// Device/Application/F020_HMI_Pages/F020_PartX_Screen
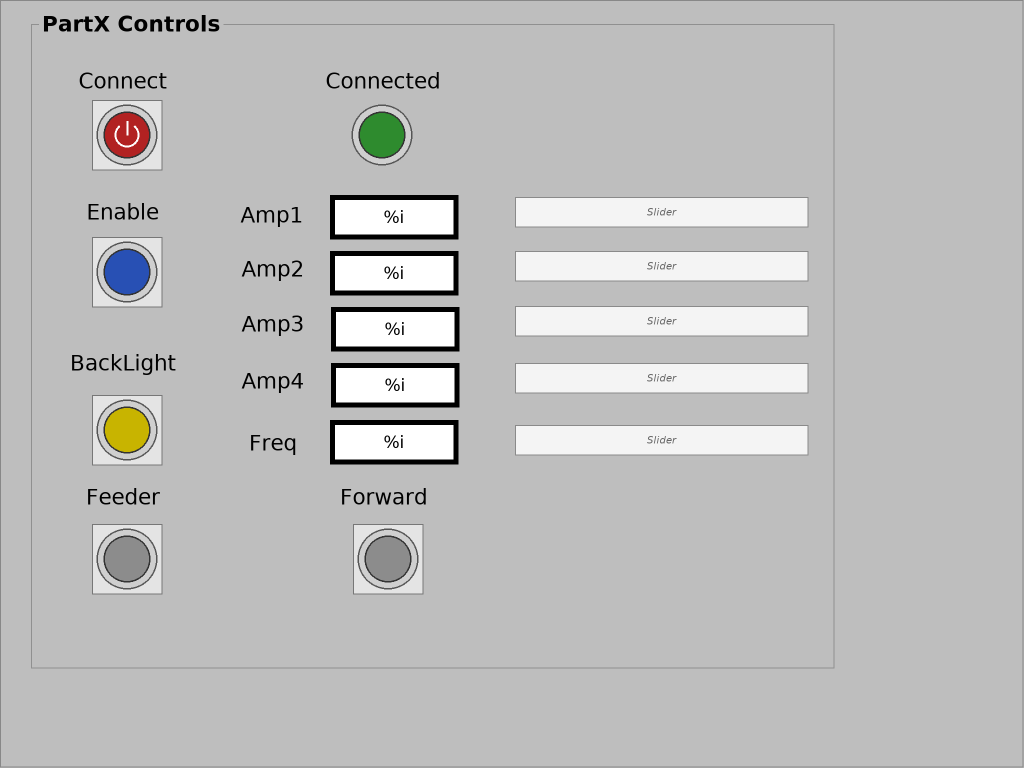
VISUALIZATION F020_PartX_Screen  // 1024x768
    GroupBox (31,16 803x652), "PartX Controls"
        Label (17,50 150x30), "Connect"
        PushSwitch (61,221 70x70), variable: GVL.PARTX.MAN, behaviour: TOGGLE, style: Switch-PushSwitch-Blue
        PowerSwitch (61,84 70x70), variable: GVL.PARTX.ENABLE_TCP, behaviour: TOGGLE, style: Switch-PowerSwitch-Red
        Label (17,181 150x30), "Enable"
        Textfield (299,179 128x44), "%i", text variable: GVL.PARTX.Amp1
            OnMouseClick: write the text variable via VisuDialogs.Numpad
        Label (277,50 150x30), "Connected"
        Label (166,184 150x30), "Amp1"
        Lamp1 (316,84 70x70), variable: F002_SR02_SOCKET_CLIENT.Client.xActive, style: Lamp-Lamp1-Green
        Textfield (299,235 128x44), "%i", text variable: GVL.PARTX.Amp2
            OnMouseClick: write the text variable via VisuDialogs.Numpad
        PushSwitch (61,379 70x70), variable: GVL.PARTX.BackLight, behaviour: TOGGLE, style: Switch-PushSwitch-Yellow
        Label (17,332 150x30), "BackLight"
        Label (167,238 150x30), "Amp2"
        Textfield (300,291 128x44), "%i", text variable: GVL.PARTX.Amp3
            OnMouseClick: write the text variable via VisuDialogs.Numpad
        Label (167,293 150x30), "Amp3"
        Textfield (300,347 128x44), "%i", text variable: GVL.PARTX.Amp4
            OnMouseClick: write the text variable via VisuDialogs.Numpad
        Label (167,350 150x30), "Amp4"
        Textfield (299,404 128x44), "%i", text variable: GVL.PARTX.Freq
            OnMouseClick: write the text variable via VisuDialogs.Numpad
        Label (167,412 150x30), "Freq"
        PushSwitch (61,508 70x70), variable: GVL.PARTX.Feeder_Enable, behaviour: TOGGLE, style: Switch-PushSwitch-Gray
        Label (17,466 150x30), "Feeder"
        Slider (484,181 293x30), variable: GVL.PARTX.Amp1, scale 0..100
        Slider (484,235 293x30), variable: GVL.PARTX.Amp2, scale 0..100
        Slider (484,290 293x30), variable: GVL.PARTX.Amp3, scale 0..100
        Label (278,466 150x30), "Forward"
        Label (472,466 150x30)
    Slider (515,363 293x30), variable: GVL.PARTX.Amp4, scale 0..100
    Slider (515,425 293x30), variable: GVL.PARTX.Freq, scale 0..100
    PushSwitch (353,524 70x70), variable: GVL.PARTX.FWD, behaviour: TOGGLE, style: Switch-PushSwitch-Gray
END_VISUALIZATION

// Device/Application/F020_HMI_Pages/Visualization
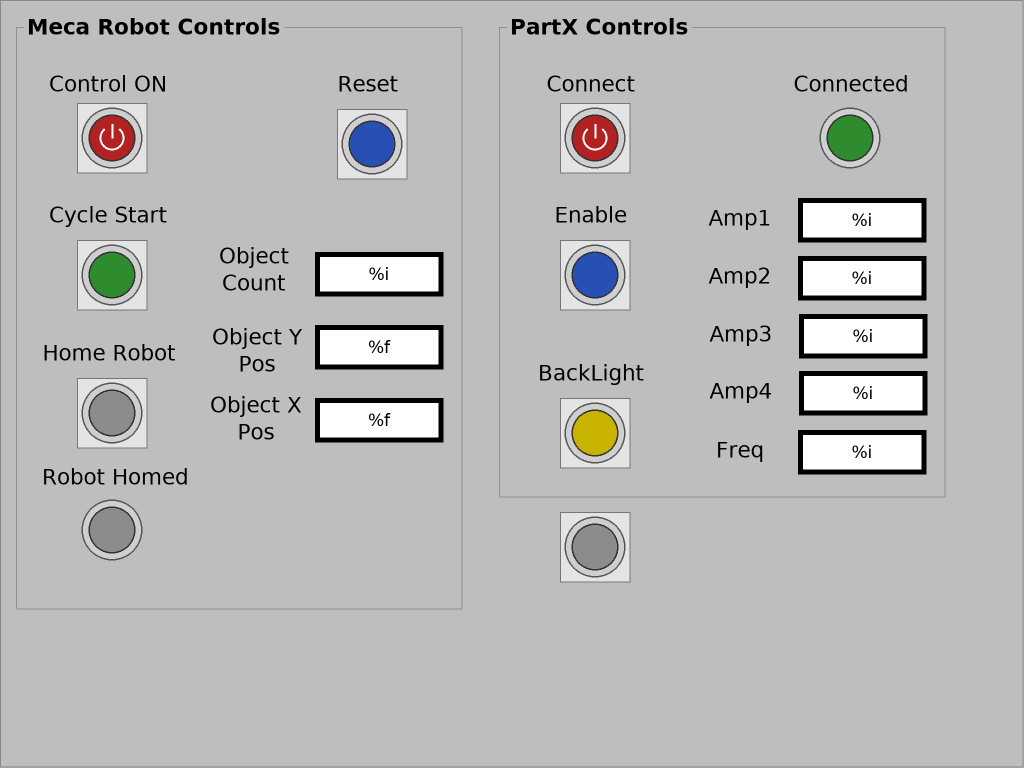
VISUALIZATION Visualization  // 1024x768
    GroupBox (16,19 446x590), "Meca Robot Controls"
        Label (17,50 150x30), "Control ON"
        PushSwitch (61,221 70x70), variable: GVL.SYS.CYCLE_START, behaviour: TAP, style: Switch-PushSwitch-Green
        PowerSwitch (61,84 70x70), variable: GVL.SYS.CONTROL_ON, behaviour: TOGGLE, style: Switch-PowerSwitch-Red
        Label (17,181 150x30), "Cycle Start"
        Textfield (299,233 128x44), "%i", text variable: GVL.CAM_1.RESULT_COUNT
        Label (163,221 150x59), "Object Count"
        Label (277,50 150x30), "Reset"
        PushSwitch (321,90 70x70), variable: GVL.SYS.RESET, behaviour: TAP, style: Switch-PushSwitch-Blue
        Label (165,369 150x61), "Object X Pos"
        Label (166,305 150x53), "Object Y Pos"
        Textfield (299,379 128x44), "%f", text variable: GVL.CAM_1.RESULT_POSX
        Textfield (299,306 128x44), "%f", text variable: GVL.CAM_1.RESULT_POSY
        Label (18,319 150x30), "Home Robot"
        PushSwitch (61,359 70x70), variable: GVL.SYS.HOME_RBT, behaviour: TAP, style: Switch-PushSwitch-Gray
        Lamp1 (61,476 70x70), variable: GVL.Meca500_1.Inputs.Status.RobotStatus.Homed, style: Lamp-Lamp1-Gray
        Label (25,443 149x30), "Robot Homed"
    GroupBox (499,19 446x478), "PartX Controls"
        Label (17,50 150x30), "Connect"
        PushSwitch (61,221 70x70), variable: GVL.PARTX.MAN, behaviour: TOGGLE, style: Switch-PushSwitch-Blue
        PowerSwitch (61,84 70x70), variable: GVL.PARTX.ENABLE_TCP, behaviour: TOGGLE, style: Switch-PowerSwitch-Red
        Label (17,181 150x30), "Enable"
        Textfield (299,179 128x44), "%i", text variable: GVL.PARTX.Amp1
            OnMouseClick: write the text variable via VisuDialogs.Numpad
        Label (277,50 150x30), "Connected"
        Label (166,184 150x30), "Amp1"
        Lamp1 (316,84 70x70), variable: F002_SR02_SOCKET_CLIENT.Client.xActive, style: Lamp-Lamp1-Green
        Textfield (299,237 128x44), "%i", text variable: GVL.PARTX.Amp2
            OnMouseClick: write the text variable via VisuDialogs.Numpad
        PushSwitch (61,379 70x70), variable: GVL.PARTX.BackLight, behaviour: TOGGLE, style: Switch-PushSwitch-Yellow
    Label (665,261 150x30), "Amp2"
    Textfield (799,314 128x44), "%i", text variable: GVL.PARTX.Amp3
        OnMouseClick: write the text variable via VisuDialogs.Numpad
    Label (666,319 150x30), "Amp3"
    Textfield (799,371 128x44), "%i", text variable: GVL.PARTX.Amp4
        OnMouseClick: write the text variable via VisuDialogs.Numpad
    Label (666,376 150x30), "Amp4"
    Textfield (798,430 128x44), "%i", text variable: GVL.PARTX.Freq
        OnMouseClick: write the text variable via VisuDialogs.Numpad
    Label (665,435 150x30), "Freq"
    Label (516,358 150x30), "BackLight"
    PushSwitch (560,512 70x70), variable: GVL.PARTX.Feeder_Enable, behaviour: TOGGLE, style: Switch-PushSwitch-Gray
END_VISUALIZATION

(* text list TL_Directions (id | default)
  0 | IDLE
  1 | Forward
  2 | Reverse
  3 | IDLE_Trigger
  4 | Bounce
   |  *)
